(* IEC 61131-3 sources: mect_apps/TP1043_01_A/Monitoring/plc, 1 file *)

(* ---- Crosstable.gvl ---- *)
VAR_GLOBAL
	Pmax AT %IW0.4:UINT;	(* PRMS phase 1 (max) *)
	EM_Firmware AT %IW0.776:UINT;	(* Firmware-Version *)
	Status AT %IW0.784:UINT;	(* Status *)
	Timeout AT %IW0.788:UINT;	(* Timeout Modbus *)
	Indirizzo AT %QW0.792:UINT;	(* Indirizzo Modbus *)
	Errore AT %IW0.796:UINT;	(* Errore Registro *)
	unused_25 AT %IW0.800:UINT;
	unused_26 AT %IW0.804:UINT;
	Ttotal AT %ID0.808:UDINT;	(* WT1 totale Contatore energia Totale Tariffa 1 *)
	Tpart AT %QD0.812:UDINT;	(* WT1 parziale Contatore energia Parziale Tariffa 1 *)
	unused_31 AT %IW0.816:UINT;
	unused_32 AT %IW0.820:UINT;
	unused_33 AT %IW0.824:UINT;
	unused_34 AT %IW0.828:UINT;
	U AT %IW0.832:UINT;	(* URMS phase 1 *)
	I AT %IW0.836:UINT;	(* IRMS phase 1 *)
	P AT %IW0.840:UINT;	(* PRMS phase 1 *)
	Q AT %IW0.844:INT;	(* QRMS phase 1 *)
	C AT %IW0.848:INT;	(* cos phi phase 1 *)
	TCP_U AT %QW0.4004:UINT;	(* URMS phase 1 *)
	TCP_I AT %QW0.4008:UINT;	(* IRMS phase 1 *)
	TCP_P AT %QW0.4012:UINT;	(* PRMS phase 1 *)
	TCP_Q AT %QW0.4016:INT;	(* QRMS phase 1 *)
	TCP_C AT %QW0.4020:INT;	(* cos phi phase 1 *)
	TCP_Pmax AT %QW0.4024:UINT;	(* PRMS phase 1 (max) *)
	TCP_Ttotal AT %QD0.4028:UDINT;	(* WT1 totale Contatore energia Totale Tariffa 1 *)
	TCP_Tpart AT %QD0.4032:UDINT;	(* WT1 parziale Contatore energia Parziale Tariffa 1 *)
	TCP_UPTIME_s AT %QD0.4036:UDINT;
	TCP_HH_MM AT %QW0.4040:UINT;
	SRV_EP_heartbeat AT %QW0.8000:UINT;	(* TCPS_STATUS NODE_09_STATUS *)
	SRV_EP_enabled_wattmeters AT %QW0.8004:UINT;	(* 0 .. 12 *)
	SRV_EP_wattmeter01_U AT %QW0.8008:INT;	(* xxx.xx V *)
	SRV_EP_wattmeter01_C AT %QW0.8012:INT;	(* +/- x.xxx *)
	SRV_EP_wattmeter01_Texp AT %QD0.8016:UDINT;	(* xxxxxxxxx.x kWh *)
	SRV_EP_wattmeter01_P AT %QW0.8020:INT;	(* +/- xxxx W *)
	SRV_EP_wattmeter01_Pmax AT %QW0.8024:INT;	(* +/- xxxx W *)
	SRV_EP_wattmeter01_T AT %QD0.8028:UDINT;	(* xxxxxxxxx.x kWh *)
	SRV_EP_wattmeter02_P AT %QW0.8032:INT;	(* +/- xxxx W *)
	SRV_EP_wattmeter02_Pmax AT %QW0.8036:INT;	(* +/- xxxx W *)
	SRV_EP_wattmeter02_T AT %QD0.8040:UDINT;	(* xxxxxxxxx.x kWh *)
	SRV_EP_wattmeter03_P AT %QW0.8044:INT;	(* +/- xxxx W *)
	SRV_EP_wattmeter03_Pmax AT %QW0.8048:INT;	(* +/- xxxx W *)
	SRV_EP_wattmeter03_T AT %QD0.8052:UDINT;	(* xxxxxxxxx.x kWh *)
	SRV_EP_wattmeter04_P AT %QW0.8056:INT;	(* +/- xxxx W *)
	SRV_EP_wattmeter04_Pmax AT %QW0.8060:INT;	(* +/- xxxx W *)
	SRV_EP_wattmeter04_T AT %QD0.8064:UDINT;	(* xxxxxxxxx.x kWh *)
	SRV_EP_wattmeter05_P AT %QW0.8068:INT;	(* +/- xxxx W *)
	SRV_EP_wattmeter05_Pmax AT %QW0.8072:INT;	(* +/- xxxx W *)
	SRV_EP_wattmeter05_T AT %QD0.8076:UDINT;	(* xxxxxxxxx.x kWh *)
	SRV_EP_wattmeter06_P AT %QW0.8080:INT;	(* +/- xxxx W *)
	SRV_EP_wattmeter06_Pmax AT %QW0.8084:INT;	(* +/- xxxx W *)
	SRV_EP_wattmeter06_T AT %QD0.8088:UDINT;	(* xxxxxxxxx.x kWh *)
	SRV_EP_wattmeter07_P AT %QW0.8092:INT;	(* +/- xxxx W *)
	SRV_EP_wattmeter07_Pmax AT %QW0.8096:INT;	(* +/- xxxx W *)
	SRV_EP_wattmeter07_T AT %QD0.8100:UDINT;	(* xxxxxxxxx.x kWh *)
	SRV_EP_wattmeter08_P AT %QW0.8104:INT;	(* +/- xxxx W *)
	SRV_EP_wattmeter08_Pmax AT %QW0.8108:INT;	(* +/- xxxx W *)
	SRV_EP_wattmeter08_T AT %QD0.8112:UDINT;	(* xxxxxxxxx.x kWh *)
	SRV_EP_wattmeter09_P AT %QW0.8116:INT;	(* +/- xxxx W *)
	SRV_EP_wattmeter09_Pmax AT %QW0.8120:INT;	(* +/- xxxx W *)
	SRV_EP_wattmeter09_T AT %QD0.8124:UDINT;	(* xxxxxxxxx.x kWh *)
	SRV_EP_wattmeter10_P AT %QW0.8128:INT;	(* +/- xxxx W *)
	SRV_EP_wattmeter10_Pmax AT %QW0.8132:INT;	(* +/- xxxx W *)
	SRV_EP_wattmeter10_T AT %QD0.8136:UDINT;	(* xxxxxxxxx.x kWh *)
	SRV_EP_wattmeter11_P AT %QW0.8140:INT;	(* +/- xxxx W *)
	SRV_EP_wattmeter11_Pmax AT %QW0.8144:INT;	(* +/- xxxx W *)
	SRV_EP_wattmeter11_T AT %QD0.8148:UDINT;	(* xxxxxxxxx.x kWh *)
	SRV_EP_wattmeter12_P AT %QW0.8152:INT;	(* +/- xxxx W *)
	SRV_EP_wattmeter12_Pmax AT %QW0.8156:INT;	(* +/- xxxx W *)
	SRV_EP_wattmeter12_T AT %QD0.8160:UDINT;	(* xxxxxxxxx.x kWh *)
	RTU0_TYPE_PORT AT %ID0.20000:UDINT;
	RTU0_BAUDRATE AT %ID0.20004:UDINT;
	RTU0_STATUS AT %ID0.20008:UDINT;
	RTU0_READS AT %ID0.20012:UDINT;
	RTU0_WRITES AT %ID0.20016:UDINT;
	RTU0_TIMEOUTS AT %ID0.20020:UDINT;
	RTU0_COMM_ERRORS AT %ID0.20024:UDINT;
	RTU0_LAST_ERROR AT %ID0.20028:UDINT;
	RTU0_WRITE_QUEUE AT %ID0.20032:UDINT;
	RTU0_BUS_LOAD AT %ID0.20036:UDINT;
	RTU3_TYPE_PORT AT %ID0.20080:UDINT;
	RTU3_BAUDRATE AT %ID0.20084:UDINT;
	RTU3_STATUS AT %ID0.20088:UDINT;
	RTU3_READS AT %ID0.20092:UDINT;
	RTU3_WRITES AT %ID0.20096:UDINT;
	RTU3_TIMEOUTS AT %ID0.20100:UDINT;
	RTU3_COMM_ERRORS AT %ID0.20104:UDINT;
	RTU3_LAST_ERROR AT %ID0.20108:UDINT;
	RTU3_WRITE_QUEUE AT %ID0.20112:UDINT;
	RTU3_BUS_LOAD AT %ID0.20116:UDINT;
	TCPS_TYPE_PORT AT %ID0.20200:UDINT;
	TCPS_IP_ADDRESS AT %ID0.20204:UDINT;
	TCPS_STATUS AT %ID0.20208:UDINT;
	TCPS_READS AT %ID0.20212:UDINT;
	TCPS_WRITES AT %ID0.20216:UDINT;
	TCPS_TIMEOUTS AT %ID0.20220:UDINT;
	TCPS_COMM_ERRORS AT %ID0.20224:UDINT;
	TCPS_LAST_ERROR AT %ID0.20228:UDINT;
	TCPS_WRITE_QUEUE AT %ID0.20232:UDINT;
	TCPS_BUS_LOAD AT %ID0.20236:UDINT;
	TCP0_TYPE_PORT AT %ID0.20240:UDINT;
	TCP0_IP_ADDRESS AT %ID0.20244:UDINT;
	TCP0_STATUS AT %ID0.20248:UDINT;
	TCP0_READS AT %ID0.20252:UDINT;
	TCP0_WRITES AT %ID0.20256:UDINT;
	TCP0_TIMEOUTS AT %ID0.20260:UDINT;
	TCP0_COMM_ERRORS AT %ID0.20264:UDINT;
	TCP0_LAST_ERROR AT %ID0.20268:UDINT;
	TCP0_WRITE_QUEUE AT %ID0.20272:UDINT;
	TCP0_BUS_LOAD AT %ID0.20276:UDINT;
	TCP1_TYPE_PORT AT %ID0.20280:UDINT;
	TCP1_IP_ADDRESS AT %ID0.20284:UDINT;
	TCP1_STATUS AT %ID0.20288:UDINT;
	TCP1_READS AT %ID0.20292:UDINT;
	TCP1_WRITES AT %ID0.20296:UDINT;
	TCP1_TIMEOUTS AT %ID0.20300:UDINT;
	TCP1_COMM_ERRORS AT %ID0.20304:UDINT;
	TCP1_LAST_ERROR AT %ID0.20308:UDINT;
	TCP1_WRITE_QUEUE AT %ID0.20312:UDINT;
	TCP1_BUS_LOAD AT %ID0.20316:UDINT;
	TCP2_TYPE_PORT AT %ID0.20320:UDINT;
	TCP2_IP_ADDRESS AT %ID0.20324:UDINT;
	TCP2_STATUS AT %ID0.20328:UDINT;
	TCP2_READS AT %ID0.20332:UDINT;
	TCP2_WRITES AT %ID0.20336:UDINT;
	TCP2_TIMEOUTS AT %ID0.20340:UDINT;
	TCP2_COMM_ERRORS AT %ID0.20344:UDINT;
	TCP2_LAST_ERROR AT %ID0.20348:UDINT;
	TCP2_WRITE_QUEUE AT %ID0.20352:UDINT;
	TCP2_BUS_LOAD AT %ID0.20356:UDINT;
	TCP3_TYPE_PORT AT %ID0.20360:UDINT;
	TCP3_IP_ADDRESS AT %ID0.20364:UDINT;
	TCP3_STATUS AT %ID0.20368:UDINT;
	TCP3_READS AT %ID0.20372:UDINT;
	TCP3_WRITES AT %ID0.20376:UDINT;
	TCP3_TIMEOUTS AT %ID0.20380:UDINT;
	TCP3_COMM_ERRORS AT %ID0.20384:UDINT;
	TCP3_LAST_ERROR AT %ID0.20388:UDINT;
	TCP3_WRITE_QUEUE AT %ID0.20392:UDINT;
	TCP3_BUS_LOAD AT %ID0.20396:UDINT;
	TCP4_TYPE_PORT AT %ID0.20400:UDINT;
	TCP4_IP_ADDRESS AT %ID0.20404:UDINT;
	TCP4_STATUS AT %ID0.20408:UDINT;
	TCP4_READS AT %ID0.20412:UDINT;
	TCP4_WRITES AT %ID0.20416:UDINT;
	TCP4_TIMEOUTS AT %ID0.20420:UDINT;
	TCP4_COMM_ERRORS AT %ID0.20424:UDINT;
	TCP4_LAST_ERROR AT %ID0.20428:UDINT;
	TCP4_WRITE_QUEUE AT %ID0.20432:UDINT;
	TCP4_BUS_LOAD AT %ID0.20436:UDINT;
	TCP5_TYPE_PORT AT %ID0.20440:UDINT;
	TCP5_IP_ADDRESS AT %ID0.20444:UDINT;
	TCP5_STATUS AT %ID0.20448:UDINT;
	TCP5_READS AT %ID0.20452:UDINT;
	TCP5_WRITES AT %ID0.20456:UDINT;
	TCP5_TIMEOUTS AT %ID0.20460:UDINT;
	TCP5_COMM_ERRORS AT %ID0.20464:UDINT;
	TCP5_LAST_ERROR AT %ID0.20468:UDINT;
	TCP5_WRITE_QUEUE AT %ID0.20472:UDINT;
	TCP5_BUS_LOAD AT %ID0.20476:UDINT;
	TCP6_TYPE_PORT AT %ID0.20480:UDINT;
	TCP6_IP_ADDRESS AT %ID0.20484:UDINT;
	TCP6_STATUS AT %ID0.20488:UDINT;
	TCP6_READS AT %ID0.20492:UDINT;
	TCP6_WRITES AT %ID0.20496:UDINT;
	TCP6_TIMEOUTS AT %ID0.20500:UDINT;
	TCP6_COMM_ERRORS AT %ID0.20504:UDINT;
	TCP6_LAST_ERROR AT %ID0.20508:UDINT;
	TCP6_WRITE_QUEUE AT %ID0.20512:UDINT;
	TCP6_BUS_LOAD AT %ID0.20516:UDINT;
	TCP7_TYPE_PORT AT %ID0.20520:UDINT;
	TCP7_IP_ADDRESS AT %ID0.20524:UDINT;
	TCP7_STATUS AT %ID0.20528:UDINT;
	TCP7_READS AT %ID0.20532:UDINT;
	TCP7_WRITES AT %ID0.20536:UDINT;
	TCP7_TIMEOUTS AT %ID0.20540:UDINT;
	TCP7_COMM_ERRORS AT %ID0.20544:UDINT;
	TCP7_LAST_ERROR AT %ID0.20548:UDINT;
	TCP7_WRITE_QUEUE AT %ID0.20552:UDINT;
	TCP7_BUS_LOAD AT %ID0.20556:UDINT;
	TCP8_TYPE_PORT AT %ID0.20560:UDINT;
	TCP8_IP_ADDRESS AT %ID0.20564:UDINT;
	TCP8_STATUS AT %ID0.20568:UDINT;
	TCP8_READS AT %ID0.20572:UDINT;
	TCP8_WRITES AT %ID0.20576:UDINT;
	TCP8_TIMEOUTS AT %ID0.20580:UDINT;
	TCP8_COMM_ERRORS AT %ID0.20584:UDINT;
	TCP8_LAST_ERROR AT %ID0.20588:UDINT;
	TCP8_WRITE_QUEUE AT %ID0.20592:UDINT;
	TCP8_BUS_LOAD AT %ID0.20596:UDINT;
	TCP9_TYPE_PORT AT %ID0.20600:UDINT;
	TCP9_IP_ADDRESS AT %ID0.20604:UDINT;
	TCP9_STATUS AT %ID0.20608:UDINT;
	TCP9_READS AT %ID0.20612:UDINT;
	TCP9_WRITES AT %ID0.20616:UDINT;
	TCP9_TIMEOUTS AT %ID0.20620:UDINT;
	TCP9_COMM_ERRORS AT %ID0.20624:UDINT;
	TCP9_LAST_ERROR AT %ID0.20628:UDINT;
	TCP9_WRITE_QUEUE AT %ID0.20632:UDINT;
	TCP9_BUS_LOAD AT %ID0.20636:UDINT;
	NODE_01_DEV_NODE AT %ID0.20688:UDINT;
	NODE_01_STATUS AT %ID0.20692:UDINT;
	NODE_02_DEV_NODE AT %ID0.20696:UDINT;
	NODE_02_STATUS AT %ID0.20700:UDINT;
	NODE_03_DEV_NODE AT %ID0.20704:UDINT;
	NODE_03_STATUS AT %ID0.20708:UDINT;
	NODE_04_DEV_NODE AT %ID0.20712:UDINT;
	NODE_04_STATUS AT %ID0.20716:UDINT;
	NODE_05_DEV_NODE AT %ID0.20720:UDINT;
	NODE_05_STATUS AT %ID0.20724:UDINT;
	NODE_06_DEV_NODE AT %ID0.20728:UDINT;
	NODE_06_STATUS AT %ID0.20732:UDINT;
	NODE_07_DEV_NODE AT %ID0.20736:UDINT;
	NODE_07_STATUS AT %ID0.20740:UDINT;
	NODE_08_DEV_NODE AT %ID0.20744:UDINT;
	NODE_08_STATUS AT %ID0.20748:UDINT;
	NODE_09_DEV_NODE AT %ID0.20752:UDINT;
	NODE_09_STATUS AT %ID0.20756:UDINT;
	NODE_10_DEV_NODE AT %ID0.20760:UDINT;
	NODE_10_STATUS AT %ID0.20764:UDINT;
	NODE_11_DEV_NODE AT %ID0.20768:UDINT;
	NODE_11_STATUS AT %ID0.20772:UDINT;
	NODE_12_DEV_NODE AT %ID0.20776:UDINT;
	NODE_12_STATUS AT %ID0.20780:UDINT;
	NODE_13_DEV_NODE AT %ID0.20784:UDINT;
	NODE_13_STATUS AT %ID0.20788:UDINT;
	NODE_14_DEV_NODE AT %ID0.20792:UDINT;
	NODE_14_STATUS AT %ID0.20796:UDINT;
	NODE_15_DEV_NODE AT %ID0.20800:UDINT;
	NODE_15_STATUS AT %ID0.20804:UDINT;
	NODE_16_DEV_NODE AT %ID0.20808:UDINT;
	NODE_16_STATUS AT %ID0.20812:UDINT;
	PLC_time AT %ID0.21560:REAL;	(* Seconds since boot (reset each 24h) *)
	PLC_timeMin AT %ID0.21564:REAL;	(* 10 seconds window start *)
	PLC_timeMax AT %ID0.21568:REAL;	(* 10 seconds window stop *)
	PLC_timeWin AT %QD0.21572:REAL;	(* Graph display window *)
	PLC_Version AT %IW0.21576:UINT;	(* Run Time version *)
	PLC_EngineStatus AT %IW0.21580:UINT;	(* PLC status *)
	PLC_ResetValues AT %QX0.21584.0:BOOL;	(* Diagnostic variables reset *)
	PLC_buzzerOn AT %QX0.21588.0:BOOL;	(* Buzzer sound (enable = 1 disable = 0) *)
	PLC_PLC_Version AT %QW0.21592:UINT;	(* PLC application version *)
	PLC_HMI_Version AT %QW0.21596:UINT;	(* HMI application version *)
	PLC_Year AT %IW0.21640:UINT;	(* Currently year *)
	PLC_Month AT %IW0.21644:UINT;	(* Currently month *)
	PLC_Day AT %IW0.21648:UINT;	(* Currently day *)
	PLC_Hours AT %IW0.21652:UINT;	(* Currently hour *)
	PLC_Minutes AT %IW0.21656:UINT;	(* Currently minutes *)
	PLC_Seconds AT %IW0.21660:UINT;	(* Currently seconds *)
	PLC_UPTIME_s AT %ID0.21664:UDINT;	(* Uptime in seconds (wraps in 136 years) *)
	PLC_UPTIME_cs AT %ID0.21668:UDINT;	(* Uptime in centiseconds = 10 ms (wraps in 497 days) *)
	PLC_WATCHDOGEN AT %QX0.21672.0:BOOL;	(* Enable Watchdog *)
	PLC_WATCHDOG_ms AT %QD0.21676:UDINT;	(* Reset Watchdog timer *)
	PLC_PRODUCT_ID AT %ID0.21680:UDINT;	(* TP/TPAC/TPLC Product ID (Hex) *)
	PLC_SERIAL_NUMBER AT %ID0.21684:UDINT;	(* TP/TPAC/TPLC Serial Number *)
	PLC_HMI_PAGE AT %QD0.21688:DINT;	(* HMI Page (page100=0x00000100) *)
	PLC_BEEP_VOLUME AT %QB0.21740:BYTE;	(* Beep volume (when buzzerOn) *)
	PLC_TOUCH_VOLUME AT %QB0.21744:BYTE;	(* Touch volume *)
	PLC_ALARM_VOLUME AT %QB0.21748:BYTE;	(* Alarm volume (when alarm) *)
	PLC_BUZZER AT %QD0.21752:UDINT;	(* Enable dynamic buzzer sound (0x44332211 up=0x11(%) on=0x22(cs) off=0x33(cs) rep=0x44(times)) *)
END_VAR
